// TIA Portal project "WordClock" (V14)

(* hardware
DEVICE "S7-1200-Station_1"  S7-1200 Station
   slot 0: "Baugruppenträger_0"  Rack  V1.0
   slot 1: "PLC"  CPU 1214C DC/DC/DC  6ES7 214-1AG40-0XB0  V4.1
   slot 3: "AQ 1x12BIT_1"  6ES7 232-4HA30-0XB0  V1.0
DEVICE "HMI"  KTP700 Basic PN
   slot 0: "HMI"  HMI  6AV2 123-2GB03-0AX0  13.0.1.0
   slot 1: "HMI_RT_1"  KTP700 Basic PN  6AV2 123-2GB03-0AX0  13.0.1.0
   slot 5: "HMI.IE_CP_1"  PROFINET Schnittstelle
      slot 1: "PROFINET Schnittstelle_1"  PROFINET Schnittstelle
         slot 1: "Port_1"  Port
*)

// ===== PLC "PLC"  CPU 1214C DC/DC/DC =====

VAR_GLOBAL   // PLC tag table "Standard-Variablentabelle"
   "System_Byte" AT %MB100 : Byte;
   "FirstScan" AT %M100.0 : Bool;
   "DiagStatusUpdate" AT %M100.1 : Bool;
   "AlwaysTRUE" AT %M100.2 : Bool;
   "AlwaysFALSE" AT %M100.3 : Bool;
   "Clock_Byte" AT %MB110 : Byte;
   "Clock_10Hz" AT %M110.0 : Bool;
   "Clock_5Hz" AT %M110.1 : Bool;
   "Clock_2.5Hz" AT %M110.2 : Bool;
   "Clock_2Hz" AT %M110.3 : Bool;
   "Clock_1.25Hz" AT %M110.4 : Bool;
   "Clock_1Hz" AT %M110.5 : Bool;
   "Clock_0.625Hz" AT %M110.6 : Bool;
   "Clock_0.5Hz" AT %M110.7 : Bool;
   "x_ES" AT %M0.0 : Bool;
   "x_IST" AT %M0.1 : Bool;
   "x_BALD" AT %M0.2 : Bool;
   "x_GLEICH" AT %M0.3 : Bool;
   "x_VIERTEL" AT %M0.4 : Bool;
   "x_ZWANZIG" AT %M0.5 : Bool;
   "x_ZEHN_Minute" AT %M0.6 : Bool;
   "x_FÜNF_Minute" AT %M0.7 : Bool;
   "x_VOR" AT %M1.0 : Bool;
   "x_NACH" AT %M1.1 : Bool;
   "x_HALB" AT %M1.2 : Bool;
   "x_ZWÖLF" AT %M1.3 : Bool;
   "x_ELF" AT %M1.4 : Bool;
   "x_ZEHN_Stunde" AT %M1.5 : Bool;
   "x_NEUN" AT %M1.6 : Bool;
   "x_ACHT" AT %M1.7 : Bool;
   "x_SIEBEN" AT %M2.0 : Bool;
   "x_SECHS" AT %M2.1 : Bool;
   "x_FÜNF_Stunde" AT %M2.2 : Bool;
   "x_VIER" AT %M2.3 : Bool;
   "x_DREI" AT %M2.4 : Bool;
   "x_ZWEI" AT %M2.5 : Bool;
   "x_EINS" AT %M2.6 : Bool;
   "x_UHR" AT %M2.7 : Bool;
   "AlleAusgänge" AT %QW0 : Word;
END_VAR

DATA_BLOCK "VersionInput"   // DB1
{ S7_Optimized_Access := 'FALSE' }
VERSION : 0.1
   VAR
      AutoTest : Bool;
      "Version" : String := 'WorkClock V2.0';
   END_VAR
BEGIN
END_DATA_BLOCK

DATA_BLOCK "DigInput"   // DB2
{ S7_Optimized_Access := 'FALSE' }
VERSION : 0.1
   VAR
      DatumUhrzeit : DTL;
   END_VAR
BEGIN
END_DATA_BLOCK

FUNCTION "DeleteMe" : Void   // FC1, FBD
{ S7_Optimized_Access := 'TRUE' }
VERSION : 0.1
   VAR_TEMP
      usi_5er_Minuten : USInt;
      usi_Stunden : USInt;
      usi_Minuten : USInt;
      usi_Sekunden : USInt;
   END_VAR
BEGIN
END_FUNCTION

FUNCTION "DatenRangieren" : Void   // FC2, SCL
{ S7_Optimized_Access := 'TRUE' }
VERSION : 0.1
   VAR_TEMP
      ErstesByte : Byte;
      ZweitesByte : Byte;
   END_VAR
BEGIN
   IF "VersionInput".AutoTest THEN
       ; //  Es werden nur die Datenbausteine verwendet  
   ELSE
       // Digitale Eingänge I0.0 - I1.7 in den Datenbaustein DigInput DB2 kopieren
       // IB0 --> DB2 Byte 0
       // IB1 --> DB2 Byte 1
       // Area 16#81 --> Input
       // Area 16#82 --> Output
       // Area 16#84 --> DB
       #ErstesByte := PEEK(area := 16#81, dbNumber := 0, byteOffset := 0);
       #ZweitesByte := PEEK(area := 16#81, dbNumber := 0, byteOffset := 1);

       POKE(area := 16#84,
            dbNumber := 2,
            byteOffset := 0,
            value := #ErstesByte);
       POKE(area := 16#84,
            dbNumber := 2,
            byteOffset := 1,
            value := #ZweitesByte);

       // DB DigOutput auf die Ausgänge Q0.0 - Q1.7 kopieren
       // DB3 Byte 0 --> QB0
       // DB3 Byte 1 --> QB1
       #ErstesByte := PEEK(area := 16#84, dbNumber := 3, byteOffset := 0);
       #ZweitesByte := PEEK(area := 16#84, dbNumber := 3, byteOffset := 1);

       POKE(area := 16#82,
            dbNumber := 0,
            byteOffset := 0,
            value := #ErstesByte);
       POKE(area := 16#82,
            dbNumber := 0,
            byteOffset := 1,
            value := #ZweitesByte);
   END_IF;
END_FUNCTION

ORGANIZATION_BLOCK "Main"   // OB1, LAD, ProgramCycle
TITLE = "Main Program Sweep (Cycle)"
{ S7_Optimized_Access := 'TRUE' }
VERSION : 0.1
   VAR_INPUT
      Initial_Call : Bool;   // Initial call of this OB
      Remanence : Bool;   // =True, if remanent data are available
   END_VAR
BEGIN

REGION Network 1: -Q1
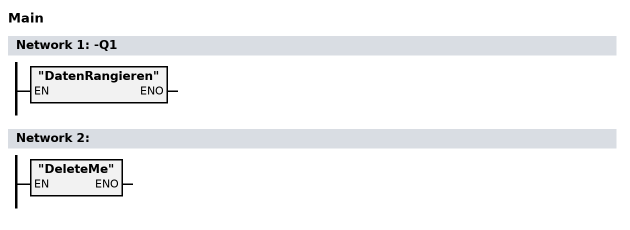
   RUNG wire#powerrail
      "DatenRangieren"()
   END_RUNG
   // the same network as SCL:
   "DatenRangieren"();
END_REGION

REGION Network 2
   RUNG wire#powerrail
      "DeleteMe"()
   END_RUNG
   // the same network as SCL:
   "DeleteMe"();
END_REGION
END_ORGANIZATION_BLOCK

ORGANIZATION_BLOCK "Startup"   // OB100, SCL, Startup
TITLE = "Complete Restart"
{ S7_Optimized_Access := 'TRUE' }
VERSION : 0.1
   VAR_INPUT
      LostRetentive : Bool;   // True if retentive data are lost
      LostRTC : Bool;   // True if date and time are lost
   END_VAR
BEGIN
   "VersionInput".AutoTest := TRUE;

   POKE(area := 16#84,     // DB
        dbNumber := 3,     // DigOutput
        byteOffset := 0,   // Byte 0
        value := byte#0);  // löschen

   POKE(area := 16#84,     // DB
        dbNumber := 3,     // Digoutput
        byteOffset := 1,   // Byte 1
        value := byte#0);  // löschen
END_ORGANIZATION_BLOCK

(* ===== HMI "HMI_RT_1" =====
connection "HMI_Verbindung_1": ETHERNET, SMART_S7_1200_OMS

HMI tags "Standard-Variablentabelle"
   "x_ES" : Bool = PLC x_ES AT %M0.0, 1 s
   "x_IST" : Bool = PLC x_IST AT %M0.1, 1 s
   "x_BALD" : Bool = PLC x_BALD AT %M0.2, 1 s
   "x_GLEICH" : Bool = PLC x_GLEICH AT %M0.3, 1 s
   "x_VIERTEL" : Bool = PLC x_VIERTEL AT %M0.4, 1 s
   "x_ZWANZIG" : Bool = PLC x_ZWANZIG AT %M0.5, 1 s
   "x_ZEHN_Minute" : Bool = PLC x_ZEHN_Minute AT %M0.6, 1 s
   "x_FÜNF_Minute" : Bool = PLC x_FÜNF_Minute AT %M0.7, 1 s
   "x_VOR" : Bool = PLC x_VOR AT %M1.0, 1 s
   "x_NACH" : Bool = PLC x_NACH AT %M1.1, 1 s
   "x_HALB" : Bool = PLC x_HALB AT %M1.2, 1 s
   "x_ZWÖLF" : Bool = PLC x_ZWÖLF AT %M1.3, 1 s
   "x_ELF" : Bool = PLC x_ELF AT %M1.4, 1 s
   "x_ZEHN_Stunde" : Bool = PLC x_ZEHN_Stunde AT %M1.5, 1 s
   "x_NEUN" : Bool = PLC x_NEUN AT %M1.6, 1 s
   "x_ACHT" : Bool = PLC x_ACHT AT %M1.7, 1 s
   "x_SIEBEN" : Bool = PLC x_SIEBEN AT %M2.0, 1 s
   "x_SECHS" : Bool = PLC x_SECHS AT %M2.1, 1 s
   "x_FÜNF_Stunde" : Bool = PLC x_FÜNF_Stunde AT %M2.2, 1 s
   "x_VIER" : Bool = PLC x_VIER AT %M2.3, 1 s
   "x_DREI" : Bool = PLC x_DREI AT %M2.4, 1 s
   "x_EINS" : Bool = PLC x_EINS AT %M2.6, 1 s
   "x_ZWEI" : Bool = PLC x_ZWEI AT %M2.5, 1 s
   "_x_UHR" : Bool = PLC x_UHR AT %M2.7, 1 s

screen "WordClock" 800x480
   TextField "Textfeld_1" at 0,0 size 77x81; Text 'ES'
      Appearance <- "x_ES"
   TextField "Textfeld_2" at 109,0 size 102x81; Text 'IST'
      Appearance <- "x_IST"
   TextField "Textfeld_3" at 244,0 size 156x81; Text 'BALD'
      Appearance <- "x_BALD"
   TextField "Textfeld_4" at 437,0 size 221x81; Text 'GLEICH'
      Appearance <- "x_GLEICH"
   TextField "Textfeld_5" at 0,65 size 248x81; Text 'VIERTEL'
      Appearance <- "x_VIERTEL"
   TextField "Textfeld_6" at 284,65 size 283x81; Text 'ZWANZIG'
      Appearance <- "x_ZWANZIG"
   TextField "Textfeld_7" at 0,130 size 163x81; Text 'ZEHN'
      Appearance <- "x_ZEHN_Minute"
   TextField "Textfeld_8" at 198,130 size 156x81; Text 'FÜNF'
      Appearance <- "x_FÜNF_Minute"
   TextField "Textfeld_9" at 393,130 size 128x81; Text 'VOR'
      Appearance <- "x_VOR"
   TextField "Textfeld_10" at 559,130 size 167x81; Text 'NACH'
      Appearance <- "x_NACH"
   TextField "Textfeld_11" at 0,195 size 156x81; Text 'HALB'
      Appearance <- "x_HALB"
   TextField "Textfeld_12" at 190,195 size 209x81; Text 'ZWÖLF'
      Appearance <- "x_ZWÖLF"
   TextField "Textfeld_13" at 432,195 size 106x81; Text 'ELF'
      Appearance <- "x_ELF"
   TextField "Textfeld_14" at 571,195 size 163x81; Text 'ZEHN'
      Appearance <- "x_ZEHN_Stunde"
   TextField "Textfeld_15" at 0,260 size 169x81; Text 'NEUN'
      Appearance <- "x_NEUN"
   TextField "Textfeld_16" at 207,260 size 161x81; Text 'ACHT'
      Appearance <- "x_ACHT"
   TextField "Textfeld_17" at 392,260 size 218x81; Text 'SIEBEN'
      Appearance <- "x_SIEBEN"
   TextField "Textfeld_18" at 0,325 size 194x81; Text 'SECHS'
      Appearance <- "x_SECHS"
   TextField "Textfeld_19" at 224,325 size 156x81; Text 'FÜNF'
      Appearance <- "x_FÜNF_Stunde"
   TextField "Textfeld_20" at 414,325 size 143x81; Text 'VIER'
      Appearance <- "x_VIER"
   TextField "Textfeld_21" at 588,325 size 148x81; Text 'DREI'
      Appearance <- "x_DREI"
   TextField "Textfeld_22" at 0,390 size 159x81; Text 'ZWEI'
      Appearance <- "x_ZWEI"
   TextField "Textfeld_23" at 191,390 size 144x81; Text 'EINS'
      Appearance <- "x_EINS"
   TextField "Textfeld_24" at 371,390 size 130x81; Text 'UHR'
      Appearance <- "_x_UHR"
   TextField "Textfeld_25" at 73,0 size 37x81; Text 'L'
   TextField "Textfeld_27" at 204,0 size 43x81; Text 'A'
   TextField "Textfeld_28" at 394,0 size 48x81; Text 'N'
   TextField "Textfeld_29" at 651,0 size 120x81; Text 'DES'
   TextField "Textfeld_30" at 245,65 size 43x81; Text 'B'
   TextField "Textfeld_31" at 561,65 size 228x81; Text 'ERUFSS'
   TextField "Textfeld_32" at 157,130 size 43x81; Text 'C'
   TextField "Textfeld_33" at 516,130 size 47x81; Text 'U'
   TextField "Textfeld_34" at 349,130 size 48x81; Text 'H'
   TextField "Textfeld_35" at 720,130 size 79x81; Text 'LE'
   TextField "Textfeld_36" at 154,195 size 38x81; Text 'F'
   TextField "Textfeld_37" at 394,195 size 41x81; Text 'E'
   TextField "Textfeld_38" at 534,195 size 37x81; Text 'L'
   TextField "Textfeld_39" at 727,195 size 48x81; Text 'D'
   TextField "Textfeld_40" at 165,260 size 43x81; Text 'K'
   TextField "Textfeld_41" at 367,260 size 29x81; Text 'I'
   TextField "Textfeld_42" at 603,260 size 162x81; Text 'RCHE'
   TextField "Textfeld_43" at 190,325 size 37x81; Text 'L'
   TextField "Textfeld_44" at 375,325 size 41x81; Text 'E'
   TextField "Textfeld_45" at 550,325 size 43x81; Text 'K'
   TextField "Textfeld_46" at 153,390 size 45x81; Text 'R'
   TextField "Textfeld_47" at 328,390 size 50x81; Text 'O'
   TextField "Textfeld_48" at 492,390 size 265x81; Text 'TECHNIK'
   TextField "Textfeld_49" at 732,325 size 42x81; Text 'T'
*)